(* CoDeSys 2.3 export: FIXBUTTON.EXP *)

(* POU FixButton, ST *)
FUNCTION_BLOCK FixButton (*Фиксация кнопки  и сброс при повторном нажатии*)
VAR_INPUT
	bIN : BOOL;
END_VAR
VAR_OUTPUT
	bQ: BOOL;
END_VAR
VAR
	Rt : R_TRIG;
END_VAR
	Rt(CLK := bIN );

	IF Rt.q THEN
		IF NOT bQ THEN
			bQ := 1;
		ELSE
			bQ := 0;
		END_IF
	END_IF
END_FUNCTION_BLOCK
